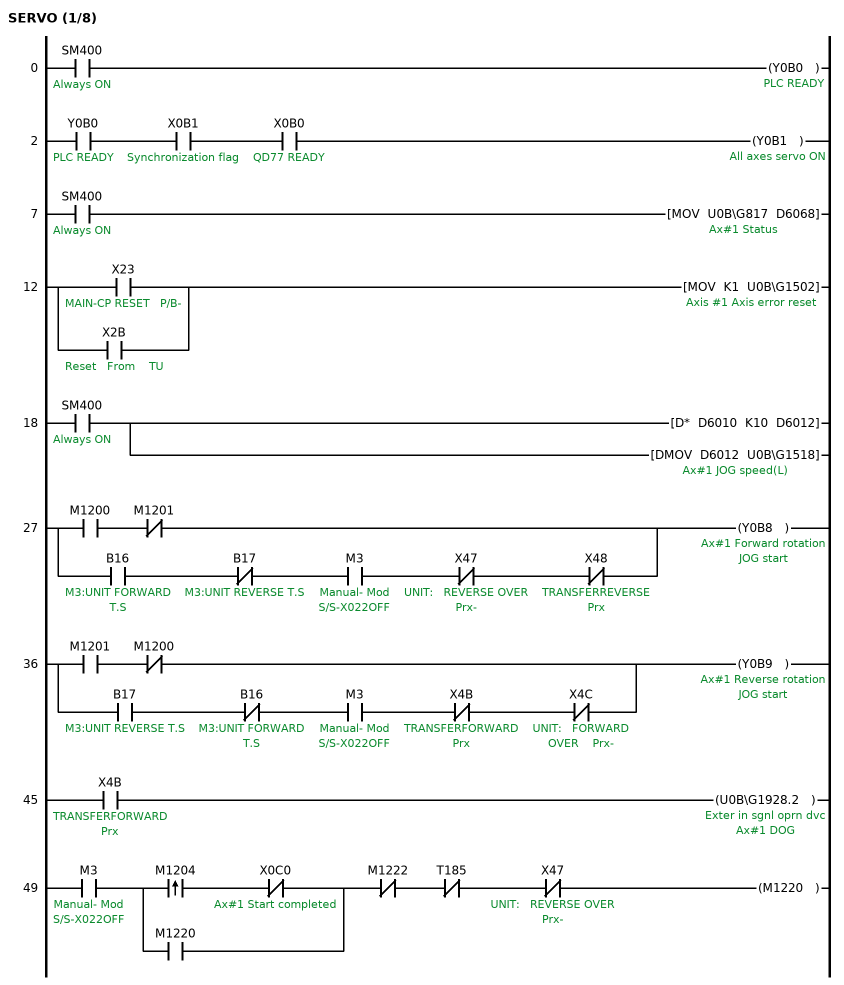
0     LD      SM400  ; Always ON
      OUT     Y0B0  ; PLC READY
2     LD      Y0B0  ; PLC READY
      AND     X0B1  ; Synchronization flag
      AND     X0B0  ; QD77 READY
      OUT     Y0B1  ; All axes servo ON
; 
7     LD      SM400  ; Always ON
      MOV     U0B\G817 D6068  ; Ax#1 Status
12    LD      X23  ; MAIN-CP RESET   P/B-
      OR      X2B  ; Reset   From    TU
      MOV     K1 U0B\G1502  ; Axis #1 Axis error reset
18    LD      SM400  ; Always ON
      D*      D6010 K10 D6012
      DMOV    D6012 U0B\G1518  ; Ax#1 JOG speed(L)
27    LD      M1200
      ANI     M1201
      LD      B16  ; M3:UNIT FORWARD T.S
      ANI     B17  ; M3:UNIT REVERSE T.S
      AND     M3  ; Manual- Mod     S/S-X022OFF
      ANI     X47  ; UNIT:   REVERSE OVER    Prx-
      ANI     X48  ; TRANSFERREVERSE Prx
      ORB
      OUT     Y0B8  ; Ax#1 Forward rotation JOG start
36    LD      M1201
      ANI     M1200
      LD      B17  ; M3:UNIT REVERSE T.S
      ANI     B16  ; M3:UNIT FORWARD T.S
      AND     M3  ; Manual- Mod     S/S-X022OFF
      ANI     X4B  ; TRANSFERFORWARD Prx
      ANI     X4C  ; UNIT:   FORWARD OVER    Prx-
      ORB
      OUT     Y0B9  ; Ax#1 Reverse rotation JOG start
45    LD      X4B  ; TRANSFERFORWARD Prx
      OUT     U0B\G1928.2  ; Exter in sgnl oprn dvc Ax#1 DOG
49    LD      M3  ; Manual- Mod     S/S-X022OFF
      LDP     M1204
      ANI     X0C0  ; Ax#1 Start completed
      OR      M1220
      ANB
      ANI     M1222
      ANI     T185
      ANI     X47  ; UNIT:   REVERSE OVER    Prx-
      OUT     M1220
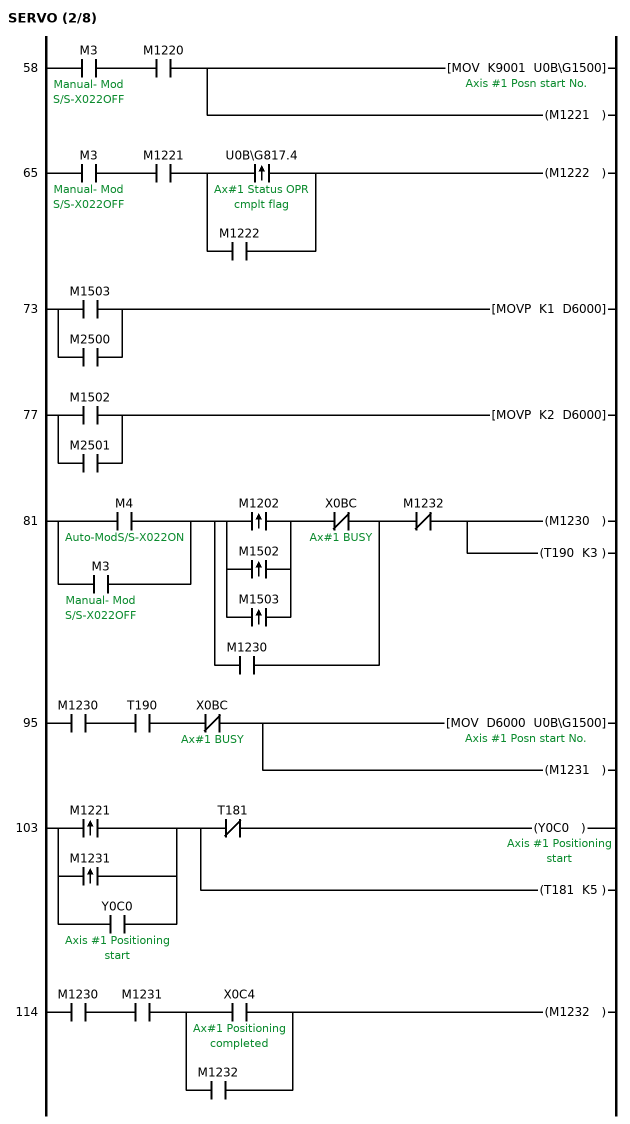
58    LD      M3  ; Manual- Mod     S/S-X022OFF
      AND     M1220
      MOV     K9001 U0B\G1500  ; Axis #1 Posn start No.
      OUT     M1221
65    LD      M3  ; Manual- Mod     S/S-X022OFF
      AND     M1221
      LDP     U0B\G817.4  ; Ax#1 Status OPR cmplt flag
      OR      M1222
      ANB
      OUT     M1222
73    LD      M1503
      OR      M2500
      MOVP    K1 D6000
77    LD      M1502
      OR      M2501
      MOVP    K2 D6000
81    LD      M4  ; Auto-ModS/S-X022ON
      OR      M3  ; Manual- Mod     S/S-X022OFF
      LDP     M1202
      ORP     M1502
      ORP     M1503
      ANI     X0BC  ; Ax#1 BUSY
      OR      M1230
      ANB
      ANI     M1232
      OUT     M1230
      OUT     T190 K3
95    LD      M1230
      AND     T190
      ANI     X0BC  ; Ax#1 BUSY
      MOV     D6000 U0B\G1500
      OUT     M1231
103   LDP     M1221
      ORP     M1231
      OR      Y0C0  ; Axis #1 Positioning start
      MPS
      ANI     T181
      OUT     Y0C0  ; Axis #1 Positioning start
      MPP
      OUT     T181 K5
114   LD      M1230
      AND     M1231
      LD      X0C4  ; Ax#1 Positioning completed
      OR      M1232
      ANB
      OUT     M1232
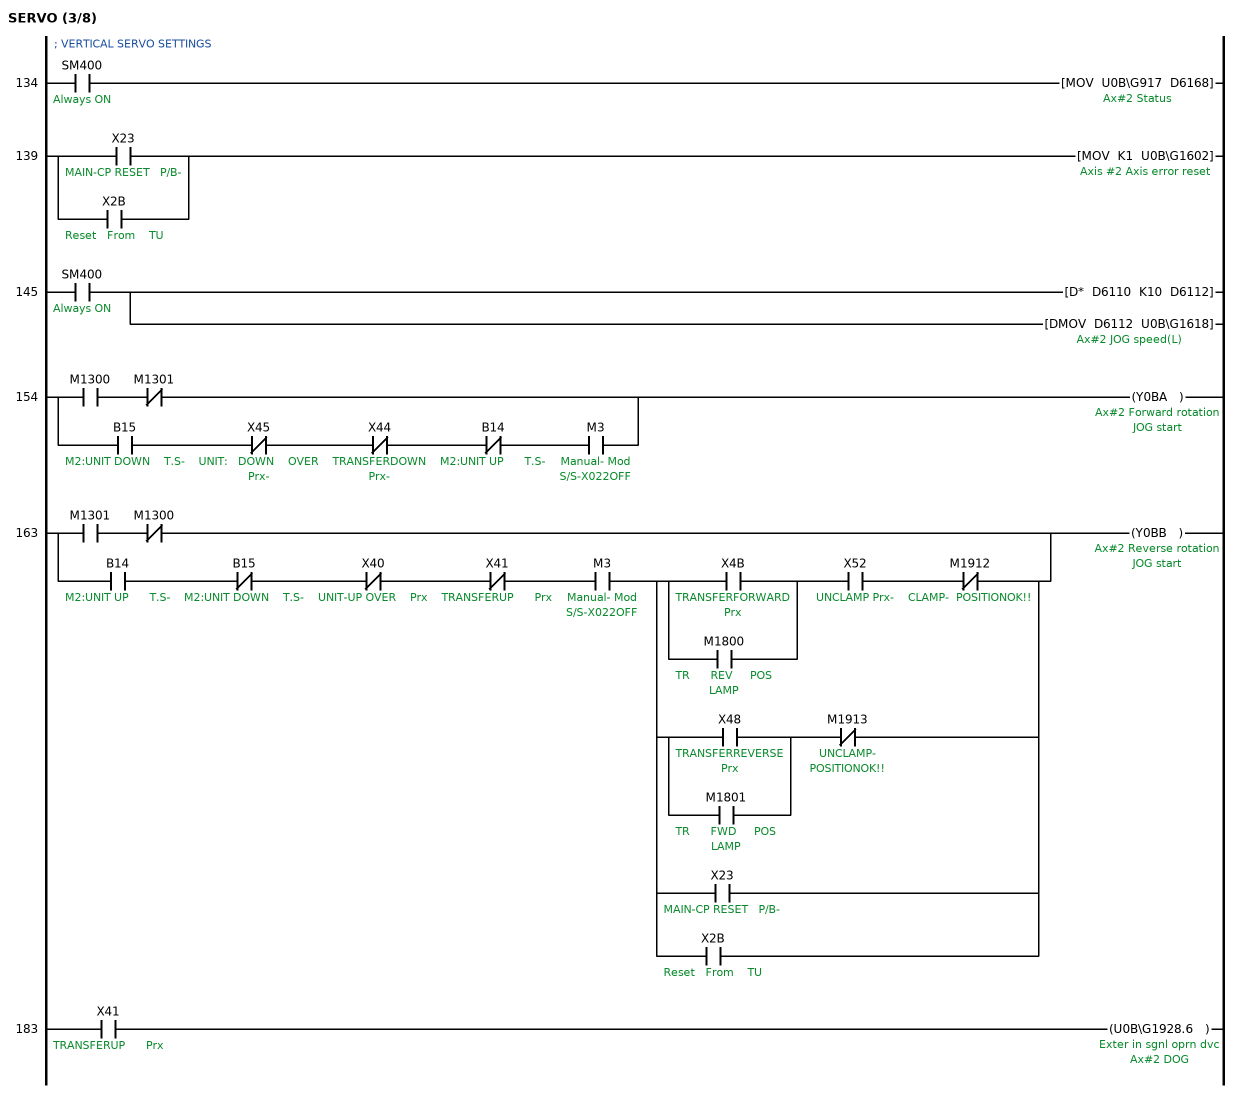
; VERTICAL SERVO SETTINGS
134   LD      SM400  ; Always ON
      MOV     U0B\G917 D6168  ; Ax#2 Status
139   LD      X23  ; MAIN-CP RESET   P/B-
      OR      X2B  ; Reset   From    TU
      MOV     K1 U0B\G1602  ; Axis #2 Axis error reset
145   LD      SM400  ; Always ON
      D*      D6110 K10 D6112
      DMOV    D6112 U0B\G1618  ; Ax#2 JOG speed(L)
154   LD      M1300
      ANI     M1301
      LD      B15  ; M2:UNIT DOWN    T.S-
      ANI     X45  ; UNIT:   DOWN    OVER    Prx-
      ANI     X44  ; TRANSFERDOWN    Prx-
      ANI     B14  ; M2:UNIT UP      T.S-
      AND     M3  ; Manual- Mod     S/S-X022OFF
      ORB
      OUT     Y0BA  ; Ax#2 Forward rotation JOG start
163   LD      M1301
      ANI     M1300
      LD      B14  ; M2:UNIT UP      T.S-
      ANI     B15  ; M2:UNIT DOWN    T.S-
      ANI     X40  ; UNIT-UP OVER    Prx
      ANI     X41  ; TRANSFERUP      Prx
      AND     M3  ; Manual- Mod     S/S-X022OFF
      LD      X4B  ; TRANSFERFORWARD Prx
      OR      M1800  ; TR      REV     POS     LAMP
      AND     X52  ; UNCLAMP Prx-
      ANI     M1912  ; CLAMP-  POSITIONOK!!
      LD      X48  ; TRANSFERREVERSE Prx
      OR      M1801  ; TR      FWD     POS     LAMP
      ANI     M1913  ; UNCLAMP-POSITIONOK!!
      ORB
      OR      X23  ; MAIN-CP RESET   P/B-
      OR      X2B  ; Reset   From    TU
      ANB
      ORB
      OUT     Y0BB  ; Ax#2 Reverse rotation JOG start
183   LD      X41  ; TRANSFERUP      Prx
      OUT     U0B\G1928.6  ; Exter in sgnl oprn dvc Ax#2 DOG
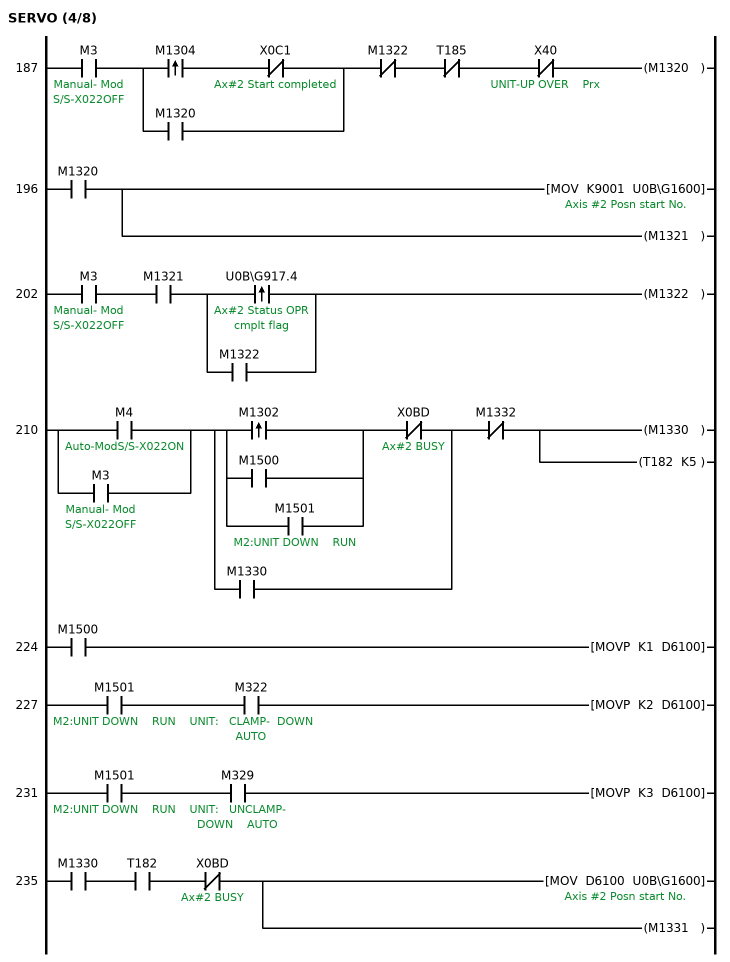
187   LD      M3  ; Manual- Mod     S/S-X022OFF
      LDP     M1304
      ANI     X0C1  ; Ax#2 Start completed
      OR      M1320
      ANB
      ANI     M1322
      ANI     T185
      ANI     X40  ; UNIT-UP OVER    Prx
      OUT     M1320
196   LD      M1320
      MOV     K9001 U0B\G1600  ; Axis #2 Posn start No.
      OUT     M1321
202   LD      M3  ; Manual- Mod     S/S-X022OFF
      AND     M1321
      LDP     U0B\G917.4  ; Ax#2 Status OPR cmplt flag
      OR      M1322
      ANB
      OUT     M1322
210   LD      M4  ; Auto-ModS/S-X022ON
      OR      M3  ; Manual- Mod     S/S-X022OFF
      LDP     M1302
      OR      M1500
      OR      M1501  ; M2:UNIT DOWN    RUN
      ANI     X0BD  ; Ax#2 BUSY
      OR      M1330
      ANB
      ANI     M1332
      OUT     M1330
      OUT     T182 K5
224   LD      M1500
      MOVP    K1 D6100
227   LD      M1501  ; M2:UNIT DOWN    RUN
      AND     M322  ; UNIT:   CLAMP-  DOWN    AUTO
      MOVP    K2 D6100
231   LD      M1501  ; M2:UNIT DOWN    RUN
      AND     M329  ; UNIT:   UNCLAMP-DOWN    AUTO
      MOVP    K3 D6100
235   LD      M1330
      AND     T182
      ANI     X0BD  ; Ax#2 BUSY
      MOV     D6100 U0B\G1600
      OUT     M1331
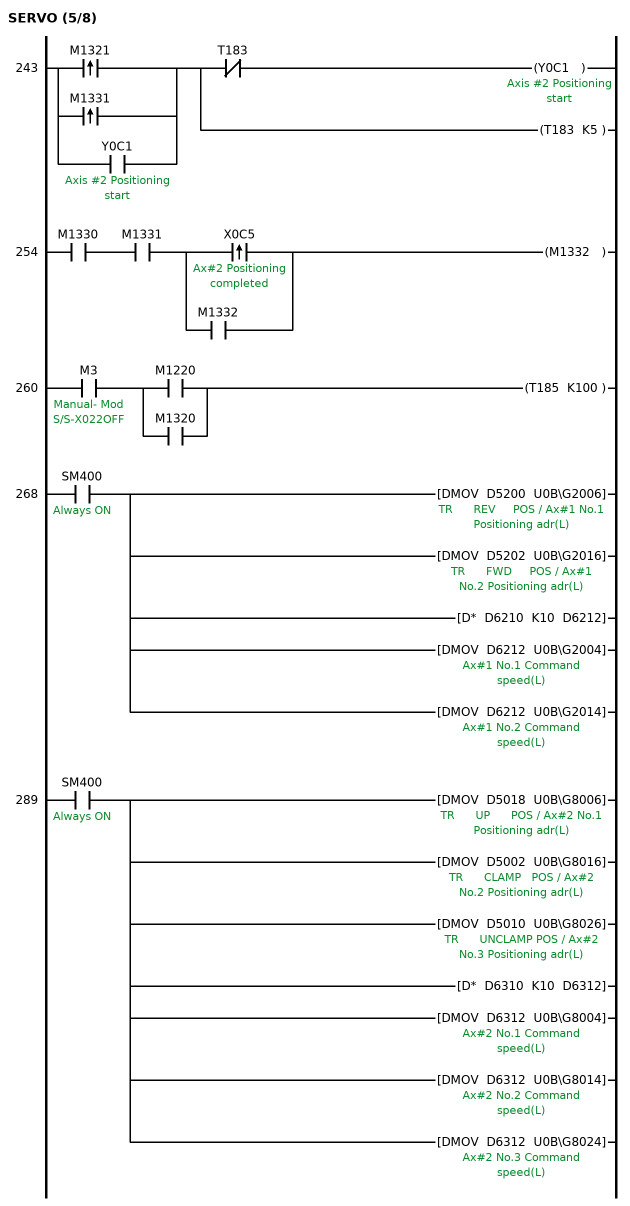
243   LDP     M1321
      ORP     M1331
      OR      Y0C1  ; Axis #2 Positioning start
      MPS
      ANI     T183
      OUT     Y0C1  ; Axis #2 Positioning start
      MPP
      OUT     T183 K5
254   LD      M1330
      AND     M1331
      LDP     X0C5  ; Ax#2 Positioning completed
      OR      M1332
      ANB
      OUT     M1332
260   LD      M3  ; Manual- Mod     S/S-X022OFF
      LD      M1220
      OR      M1320
      ANB
      OUT     T185 K100
268   LD      SM400  ; Always ON
      DMOV    D5200 U0B\G2006  ; TR      REV     POS / Ax#1 No.1 Positioning adr(L)
      DMOV    D5202 U0B\G2016  ; TR      FWD     POS / Ax#1 No.2 Positioning adr(L)
      D*      D6210 K10 D6212
      DMOV    D6212 U0B\G2004  ; Ax#1 No.1 Command speed(L)
      DMOV    D6212 U0B\G2014  ; Ax#1 No.2 Command speed(L)
289   LD      SM400  ; Always ON
      DMOV    D5018 U0B\G8006  ; TR      UP      POS / Ax#2 No.1 Positioning adr(L)
      DMOV    D5002 U0B\G8016  ; TR      CLAMP   POS / Ax#2 No.2 Positioning adr(L)
      DMOV    D5010 U0B\G8026  ; TR      UNCLAMP POS / Ax#2 No.3 Positioning adr(L)
      D*      D6310 K10 D6312
      DMOV    D6312 U0B\G8004  ; Ax#2 No.1 Command speed(L)
      DMOV    D6312 U0B\G8014  ; Ax#2 No.2 Command speed(L)
      DMOV    D6312 U0B\G8024  ; Ax#2 No.3 Command speed(L)
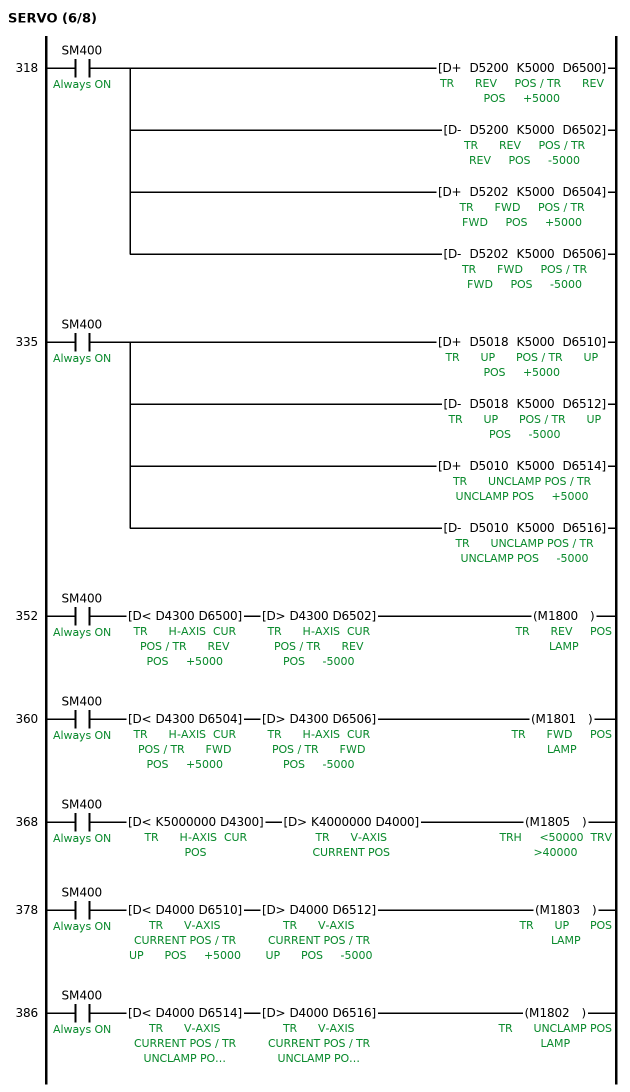
318   LD      SM400  ; Always ON
      D+      D5200 K5000 D6500  ; TR      REV     POS     +5000
      D-      D5200 K5000 D6502  ; TR      REV     POS     -5000
      D+      D5202 K5000 D6504  ; TR      FWD     POS     +5000
      D-      D5202 K5000 D6506  ; TR      FWD     POS     -5000
335   LD      SM400  ; Always ON
      D+      D5018 K5000 D6510  ; TR      UP      POS     +5000
      D-      D5018 K5000 D6512  ; TR      UP      POS     -5000
      D+      D5010 K5000 D6514  ; TR      UNCLAMP POS     +5000
      D-      D5010 K5000 D6516  ; TR      UNCLAMP POS     -5000
352   LD      SM400  ; Always ON
      ANDD<   D4300 D6500  ; TR      H-AXIS  CUR     POS / TR      REV     POS     +5000
      ANDD>   D4300 D6502  ; TR      H-AXIS  CUR     POS / TR      REV     POS     -5000
      OUT     M1800  ; TR      REV     POS     LAMP
360   LD      SM400  ; Always ON
      ANDD<   D4300 D6504  ; TR      H-AXIS  CUR     POS / TR      FWD     POS     +5000
      ANDD>   D4300 D6506  ; TR      H-AXIS  CUR     POS / TR      FWD     POS     -5000
      OUT     M1801  ; TR      FWD     POS     LAMP
368   LD      SM400  ; Always ON
      ANDD<   K5000000 D4300  ; TR      H-AXIS  CUR     POS
      ANDD>   K4000000 D4000  ; TR      V-AXIS  CURRENT POS
      OUT     M1805  ; TRH     <50000  TRV     >40000
378   LD      SM400  ; Always ON
      ANDD<   D4000 D6510  ; TR      V-AXIS  CURRENT POS / TR      UP      POS     +5000
      ANDD>   D4000 D6512  ; TR      V-AXIS  CURRENT POS / TR      UP      POS     -5000
      OUT     M1803  ; TR      UP      POS     LAMP
386   LD      SM400  ; Always ON
      ANDD<   D4000 D6514  ; TR      V-AXIS  CURRENT POS / TR      UNCLAMP POS     +5000
      ANDD>   D4000 D6516  ; TR      V-AXIS  CURRENT POS / TR      UNCLAMP POS     -5000
      OUT     M1802  ; TR      UNCLAMP POS     LAMP
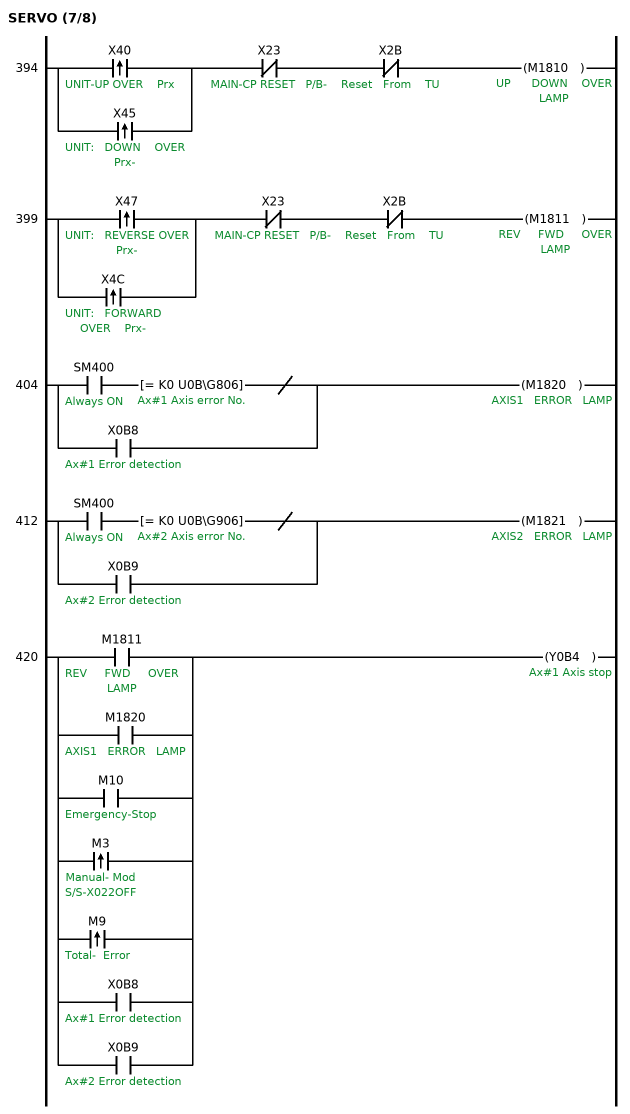
394   LDP     X40  ; UNIT-UP OVER    Prx
      ORP     X45  ; UNIT:   DOWN    OVER    Prx-
      ANI     X23  ; MAIN-CP RESET   P/B-
      ANI     X2B  ; Reset   From    TU
      OUT     M1810  ; UP      DOWN    OVER    LAMP
399   LDP     X47  ; UNIT:   REVERSE OVER    Prx-
      ORP     X4C  ; UNIT:   FORWARD OVER    Prx-
      ANI     X23  ; MAIN-CP RESET   P/B-
      ANI     X2B  ; Reset   From    TU
      OUT     M1811  ; REV     FWD     OVER    LAMP
404   LD      SM400  ; Always ON
      AND=    K0 U0B\G806  ; Ax#1 Axis error No.
      INV
      OR      X0B8  ; Ax#1 Error detection
      OUT     M1820  ; AXIS1   ERROR   LAMP
412   LD      SM400  ; Always ON
      AND=    K0 U0B\G906  ; Ax#2 Axis error No.
      INV
      OR      X0B9  ; Ax#2 Error detection
      OUT     M1821  ; AXIS2   ERROR   LAMP
420   LD      M1811  ; REV     FWD     OVER    LAMP
      OR      M1820  ; AXIS1   ERROR   LAMP
      OR      M10  ; Emergency-Stop
      ORP     M3  ; Manual- Mod     S/S-X022OFF
      ORP     M9  ; Total-  Error
      OR      X0B8  ; Ax#1 Error detection
      OR      X0B9  ; Ax#2 Error detection
      OUT     Y0B4  ; Ax#1 Axis stop
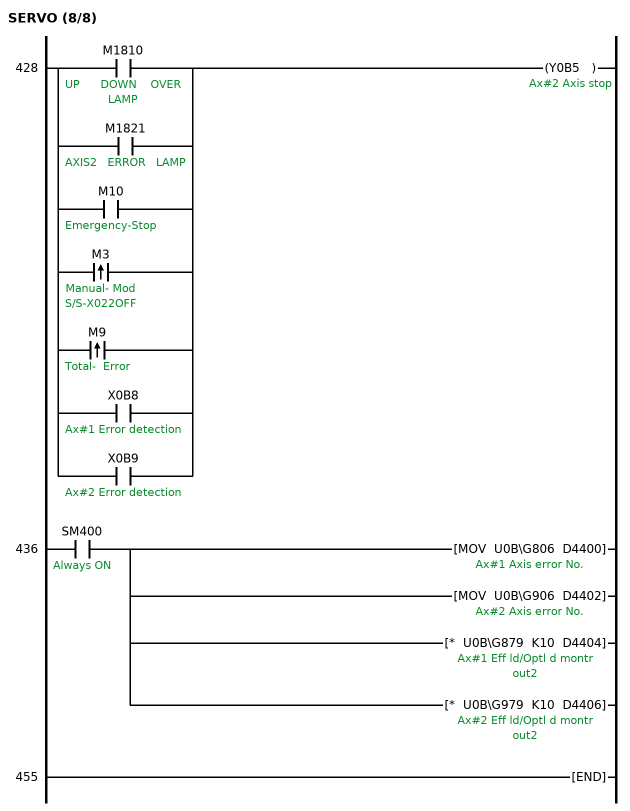
428   LD      M1810  ; UP      DOWN    OVER    LAMP
      OR      M1821  ; AXIS2   ERROR   LAMP
      OR      M10  ; Emergency-Stop
      ORP     M3  ; Manual- Mod     S/S-X022OFF
      ORP     M9  ; Total-  Error
      OR      X0B8  ; Ax#1 Error detection
      OR      X0B9  ; Ax#2 Error detection
      OUT     Y0B5  ; Ax#2 Axis stop
436   LD      SM400  ; Always ON
      MOV     U0B\G806 D4400
      MOV     U0B\G906 D4402
      *       U0B\G879 K10 D4404  ; Ax#1 Eff ld/Optl d montr out2
      *       U0B\G979 K10 D4406  ; Ax#2 Eff ld/Optl d montr out2
455   END
END_PROGRAM

// device comments not shown above
X1  ; CH1 Cntr val lrg(pt No. 1)
X2  ; CH1 Cntr val coinc(pt No. 1)
X3  ; CH1 Cntr val sml(pt No. 1)
X4  ; CH1 Extrnl prst rqst dtc
X5  ; CH1 Cntr val lrg(pt No. 2)
X6  ; CH1 Cntr val coinc(pt No. 2)
X7  ; CH1 Cntr val sml(pt No. 2)
X8  ; CH2 Cntr val lrg(pt No. 1)
X9  ; CH2 Cntr val coinc(pt No. 1)
X0A  ; CH2 Cntr val sml(pt No. 1)
X0B  ; CH2 Extrnl prst rqst dtc
X0C  ; CH2 Cntr val lrg(pt No. 2)
X0D  ; CH2 Cntr val coinc(pt No. 2)
X0E  ; CH2 Cntr val sml(pt No. 2)
X0F  ; Fuse broken detection flag
X3D  ; SLAT C/VHOME    Prx-
X3E  ; SLAT C/VCHECK   P/H-
X5A  ; FOOT S/W
X0B4  ; Ax#1 M code ON
X0B5  ; Ax#2 M code ON
X0B6  ; Ax#3 M code ON
X0B7  ; Ax#4 M code ON
X0BA  ; Ax#3 Error detection
X0BB  ; Ax#4 Error detection
X0BE  ; Ax#3 BUSY
X0BF  ; Ax#4 BUSY
X0C2  ; Ax#3 Start completed
X0C3  ; Ax#4 Start completed
X0C6  ; Ax#3 Positioning completed
X0C7  ; Ax#4 Positioning completed
X144  ; BUZZER- STOP    T.S-
M41  ; AXIS#1  UP.DOWN Error   No.
M42  ; AXIS#2  FWD.REV Error   No.
M44  ; AXIS#4  FWD.REV Error   No.
M55  ; AXIS#2-1TURNING OVER
M90  ; AXIS#1  LH.RH   M.P.G   ON
M91  ; AXIS#1  LH.RH   M.P.G   ON-SET
M92  ; AXIS#1  LH.RH   M.P.G   OFF
M127  ; Dummy   Origin
M309  ; CENTER  CHECKINGPrx-X054PLS-SET
M310  ; Auto-RunAux
M337  ; Dummy
M350  ; UNCLAMP
M391  ; PUSHER- FWD
M392  ; PUSHER- REV
M451  ; BELT C/V#1      STOP
M452  ; BELT C/V#2      RUN
M460  ; From;   Cabinet 180Turn
M1941  ; AXIS#1-4ClampingUnclamp OK!!
M1942  ; AXIS#1-4ClampingClamp   OK!!
M1951  ; AXIS#2-1Turning Origin  OK!!
M2010  ; Rotor   Nut     Check   Step10
M2011  ; Rotor   Nut     Check   Step11
M2012  ; Rotor   Nut     Check   Step12
M2013  ; Rotor   Nut     Check   Step13
M2014  ; Rotor   Nut     Check   Step14
M2015  ; Rotor   Nut     Check   Step15
B0  ; MODEL   CHANGE  T.S-
B1  ; PRODUCT COUNTER RESET   T.S-
B4  ; PRODUCT COUNTER "+"     T.S-
B5  ; PRODUCT COUNTER "-"     T.S-
B6  ; Model-Nameplate Input
B8  ; "JOG"   Low/HighSpeed   T.S-
B0C  ; STEP-MOD"+"     T.S-
B0D  ; Machine PASS-MOD
B20  ; ConveyorPusher- Fwd     T.S-
B21  ; ConveyorPusher- Rev     T.S-
B22  ; M01F    BELT C/V#1      RUN
B23  ; M01F    BELT C/V#1      STOP
B24  ; BELT C/V#2      RUN
B25  ; BELT C/V#2      STOP
B26  ; GUIDE   FWD     T.S-
B27  ; GUIDE   REV     T.S-
B30  ; CHUTTER Side-   Pusher  REV
B32  ; CHUTTER STOPPER DOWN    T.S-
B34  ; PACKING Center- Fwd     T.S-
B36  ; CHUTTER UP      T.S-
B37  ; CHUTTER DOWN    T.S-
B38  ; ConveyorStopper Down    T.S-
B3A  ; M02F    ConveyorRun     T.S-
B3C  ; CHUTTER PUSHER: FWD     T.S
B3D  ; CHUTTER PUSHER: REV     T.S
B3E  ; GUIDE   FWD     T.S-
B3F  ; GUIDE   REV     T.S-
B41  ; AXIS#4  Forward ClampãÁ AUX
B42  ; AXIS#4  Forward UnclampãÁAUX
B0A3  ; AXIS#1-2Forward ClampãÁ AUX
B132  ; CHUTTER STOPPER Up      Lamp
B138  ; ConveyorStopper UP      Lamp
B151  ; Axis#1-1Up.Down Clamp-  Input
B152  ; Axis#1-1Up.Down Unclamp-Input
B154  ; Axis#1-1UP.DOWN "+" JOG T.S-
B155  ; Axis#1-1UP.DOWN "-" JOG T.S-
B161  ; Axis#1-2Forward Clamp   Input
B162  ; Axis#1-2Forward Unclamp Input
B164  ; Axis#1-2FWD.REV "+" JOG T.S-
B165  ; Axis#1-2FWD.REV "-" JOG T.S-
B171  ; Axis#1-3Left    Input
B172  ; Axis#1-3Right   Input
B174  ; Axis#1-3LH.RH   "+" JOG  T.S-
B175  ; Axis#1-3LH.RH   "-" JOG  T.S-
B180  ; Axis#1-4ClampingOrigin  T.S-
B181  ; Axis#1-4Clamp   Input   T.S-
B184  ; Axis#1-4CLAMPING"+" JOG T.S-
B185  ; Axis#4  Reverse JOG     T.S-
B190  ; Axis#2-1Turn ingOrigin  T.S-
B191  ; Axis#2-1Turn    Input
B192  ; Axis#2-1Return  Input
B194  ; AXIS#2-1TURNING "+"JOG  T.S-
B195  ; AXIS#2-1TURNING "-"JOG  T.S-
Y0  ; CH1 Coinc sgnl No. 1 rst cmd
Y1  ; CH1 Preset command
Y2  ; CH1 Coinc sgnl enbl cmd
Y3  ; CH1 Down count command
Y5  ; CH1 Extrnl prst dtc rst cmd
Y6  ; CH1 Cntr fnctn sel strt cmd
Y7  ; CH1 Coinc sgnl No. 2 rst cmd
Y8  ; CH2 Coinc sgnl No. 1 rst cmd
Y9  ; CH2 Preset command
Y0A  ; CH2 Coinc sgnl enbl cmd
Y0B  ; CH2 Down count command
Y0C  ; CH2 Count enable command
Y0D  ; CH2 Extrnl prst dtc rst cmd
Y0E  ; CH2 Cntr fnctn sel strt cmd
Y0F  ; CH2 Coinc sgnl No. 2 rst cmd
Y63  ; AXIS#1-4ClampingDOG     Prx-X051
Y64  ; AXIS#2-1Turn.   Return  DOG-X052
Y0B6  ; Ax#3 Axis stop
Y0B7  ; Ax#4 Axis stop
Y0BC  ; Ax#3 Forward rotation JOG start
Y0BD  ; Ax#3 Reverse rotation JOG start
Y0BE  ; Ax#4 Forward rotation JOG start
Y0BF  ; Ax#4 Reverse rotation JOG start
Y0C2  ; Axis #3 Positioning start
Y0C3  ; Axis #4 Positioning start
Y0C4  ; Ax#1 Execution prohibition flag
Y0C5  ; Ax#2 Execution prohibition flag
Y0C6  ; Ax#3 Execution prohibition flag
Y0C7  ; Ax#4 Execution prohibition flag
T400  ; NORMAL- ON
T498  ; Model-Nameplate Input
T499  ; MODEL-  CHANGE  T.S-B000
T500  ; MODEL-  CHANGE  T.S-B000
T501  ; Axis#1-1Up.Down Clamp-  T.S-B151
T502  ; Axis#1-1Up.Down Unclamp T.S-B152
T503  ; Axis#1-2Forward Clamp   T.S-B161
T504  ; Axis#1-2Forward Unclamp T.S-B162
T505  ; Axis#1-3Left    Input   T.S-B171
T506  ; Axis#1-3Right   Input   T.S-B172
T507  ; Axis#1-4Clamp   Input   T.S-B181
T509  ; Axis#2-1Turn    Input   T.S-B191
T510  ; Axis#2-1Return  Input   T.S-B192
T514  ; Axis#1-4ClampingOrigin  T.S-B180
T515  ; Axis#2-1Turn ingOrigin  T.S-B190
T524  ; PRODUCT COUNTER "+"     T.S-B004
T525  ; PRODUCT COUNTER "-"     T.S-B005
L4  ; Axis#1-4ClampingOrigin  T.S-
L5  ; Axis#2-1Turn ingOrigin  T.S-B190
L40  ; AXIS#1-4ClampingUnclamp-RUN
L41  ; AXIS#1-4ClampingClamp-  RUN
L42  ; AXIS#4  Forward UnclampãÁRUN
L50  ; AXIS#2-1Turning Return  RUN
L51  ; AXIS#2-1Turning Turn    RUN
D8  ; TOUCH-  SCREEN  CHANGE
D90  ; AXIS#1  MPG-ÛÃáÜDouble- speed
D92  ; AXIS#1  MPG     K1=úÉÊ¦ K=0ÜôÊ¦
D1008  ; Password
D1100  ; AXIS#1-1UP.DOWN Present-Value
D1120  ; AXIS#1-1Up.Down Clamp-  Position
D1124  ; Axis#1-1Up.Down Clamp-  DATA
D1134  ; Axis#1-1Up.Down Unclamp DATA
D1224  ; Axis#1-2Forward Clamp   DATA
D1234  ; Axis#1-2Forward Unclamp DATA
D1324  ; Axis#1-3LH.RH   Left    DATA
D1334  ; Axis#1-3LH.RH   Right   DATA
D1400  ; AXIS#1-4ClampingPresent-Value
D1404  ; AXIS#1-4ClampingError   No.
D1408  ; Axis#1-4ClampingLoad-   Torque(%
D1420  ; Axis#1-4Clamp   PositionData
D1424  ; Axis#1-4Clamp   DATA
D1444  ; ClampingUnclamp D1400 - K0
D1448  ; ClampingClamp   D1400 - D1420
D1500  ; AXIS#2-1Turning Present-Value
D1504  ; AXIS#2-1Turning Error   No.
D1508  ; Axis#2-1Turning Load-   Torque(%
D1520  ; AXIS#2-1Turning PositionData
D1524  ; Axis#2-1Turn    DATA
D1530  ; AXIS#2-1Return  PositionData
D1534  ; Axis#2-1Return  DATA
D1544  ; AXIS#2-1Turning D1500 - K0
D1548  ; Turning PositionD1500 - D1520
D1552  ; Return  PositionD1500 - D1530
D4004  ; AXIS#1-1LH.RH   Error   No.
D4008  ; Axis#1-1LH.RH   Load-   Torque(%
D4032  ; AXIS#1-1UP.DOWN ACC.
D4036  ; AXIS#1-1UP.DOWN DEC.
D4040  ; Axis#1-1LH.RH   JOG     Speed
D5014  ; AXIS#1-1LH.RH   RIGHT   SPEED
D6200  ; TR      REV     POS
D6202  ; TR      FWD     POS
R0  ; MODEL   No.
R1  ; MODEL   No.     WRITE
R16  ; FROM;KEYLH.RH   Left
R22  ; Axis#1-1UP      SPEED-  DATA
R70  ; Axis#1-4ClampingJOG-Low Speed
R74  ; Axis#1-4ClampingJOG-HighSpeed
R78  ; AXIS#1-4Clamp   SPEED-  DATA
R82  ; AXIS#1-4Unclamp SPEED-  DATA
R90  ; Axis#2-1Turning JOG-Low Speed
R94  ; Axis#2-1TurningJOG-HighSpeed
R208  ; AXIS#1-1LH.RH   Upper-  Limit
R212  ; AXIS#1-1LH.RH   Lower-  Limit
R216  ; Axis#1-2Up.Down Speed   Override
R230  ; LH.RH   SV#4(1-4Current Value
R236  ; Axis#1-2Fwd,Rev Speed   Override
R256  ; Axis#1-3LH.RH   Speed   Override
R260  ; AXIS#1-4ClampingACC.
R264  ; AXIS#1-4ClampingDEC.
R268  ; AXIS#1-4ClampingUpper-  Limit
R272  ; AXIS#1-4ClampingLower-  Limit
R276  ; Axis#1-4ClampingSpeed   Override
R280  ; AXIS#2-1Turning ACC.
R284  ; AXIS#2-1Turning DEC.
R288  ; AXIS#2-1Turning Upper-  Limit
R292  ; AXIS#2-1Turning Lower-  Limit
R296  ; Axis#2-1TurniingSpeed   Override
R900  ; ModelÜ¬-Nameplate       Display
R920  ; ModelÜ¬-Nameplate       Input
R1000  ; Model   No._ _  Data-   Storage
R1100  ; AXIS#1-3UP.DOWN CLAMPÁöÁ¡
R1200  ; AXIS#1-3UP.DOWN UNCLAMP ÁöÁ¡
R1300  ; AXIS#1-4LH.RH   Left
R1500  ; AXIS#1-1Up.Down Unclamp-Storage
R2000  ; Axis#1-2Forward Clamp-  Storage
R2500  ; Axis#1-2Forward Unclamp-Storage
R3000  ; Axis#1-3Left-   Storage
R3500  ; Axis#1-3Right-  Storage
R4000  ; Axis#1-4Clamp   Storage
R5000  ; Axis#2-1Turn-   Storage
R5500  ; Axis#2-1Return- Storage
R10000  ; ModelÜ¬-Nameplate       Storage
